// TIA Portal V15.1 export
// export: Created 2024-06-21T08:40:43.8980344Z, ExportSetting WithDefaults, DisplayName Totally Integrated Automation Portal, DisplayVersion V15.1 Update 5, DisplayName TIA Portal Openness, DisplayVersion V15.1 Update 5, DisplayName SINAMICS Startdrive Advanced, DisplayVersion V15.1, DisplayName G130, G150, S120, S150, SINAMICS MV, S210, DisplayVersion V15.1, DisplayName G110M, G120, G120C, G120D, G120P, DisplayVersion V15.1, DisplayName STEP 7 Professional, DisplayVersion V15.1 Update 5, DisplayName STEP 7 Safety, DisplayVersion V15.1, DisplayName WinCC Professional, DisplayVersion V15.1 Update 5, DisplayName SIMATIC Visualization Architect, DisplayVersion V15.1
DATA_BLOCK "_209210ZS01AEAK"   // DB321
{ S7_Optimized_Access := 'FALSE' }
AUTHOR : VCC
VERSION : 0.1
// stored: AutoNumber false, DBAccessibleFromOPCUA true, IsOnlyStoredInLoadMemory false, IsWriteProtectedInAS false
   VAR RETAIN
      AB_AK01E1QM10 { ExternalAccessible := 'False'; ExternalVisible := 'False'; ExternalWritable := 'False'} : Bool;   // 400VAC - Overload protection MoviDrive chain Mode Zone 210
      AB_AK01E1QM11 { ExternalAccessible := 'False'; ExternalVisible := 'False'; ExternalWritable := 'False'} : Bool;   // 400VAC - Overload protection MoviFit chain Mode Zone 210
      AB_AK03E1QM130 { ExternalAccessible := 'False'; ExternalVisible := 'False'; ExternalWritable := 'False'} : Bool;   // 400VAC - Overload protection Brake Resistor 209210CR21
      AB_AK03E1QM133 { ExternalAccessible := 'False'; ExternalVisible := 'False'; ExternalWritable := 'False'} : Bool;   // 400VAC - Overload protection Brake Resistor 209210CR23
      AA_AE01E3FS07_CH1 { ExternalAccessible := 'False'; ExternalVisible := 'False'; ExternalWritable := 'False'} : Bool;   // 24VDC Fuse - ModeZone210 - Switch / Busnode 210AX01 & 210AS10
      AA_AE01E3FS07_CH2 { ExternalAccessible := 'False'; ExternalVisible := 'False'; ExternalWritable := 'False'} : Bool;   // 24VDC Fuse - ModeZone210 - Busnode 210AX02 & 210AS11 & 210AS20
      AC_AE01E3FS08_CH1 { ExternalAccessible := 'False'; ExternalVisible := 'False'; ExternalWritable := 'False'} : Bool;   // 24VDC Fuse - ModeZone210 - RFID Reader
      AA_AE01E3FS08_CH2 { ExternalAccessible := 'False'; ExternalVisible := 'False'; ExternalWritable := 'False'} : Bool;   // 24VDC Fuse - ModeZone210 - Eco Modules
      AD_AE01E3FS07_CH1 { ExternalAccessible := 'False'; ExternalVisible := 'False'; ExternalWritable := 'False'} : Bool;   // 24VDC Fuse - ModeZone210 - Switch / Busnode 210AX01 & 210AS10
      AD_AE01E3FS07_CH2 { ExternalAccessible := 'False'; ExternalVisible := 'False'; ExternalWritable := 'False'} : Bool;   // 24VDC Fuse - ModeZone210 - Busnode 210AX02 & 210AS11 & 210AS20
      AD_AE01E3FS08_CH1 { ExternalAccessible := 'False'; ExternalVisible := 'False'; ExternalWritable := 'False'} : Bool;   // 24VDC Fuse - ModeZone210 - RFID Reader
      AD_AE01E3FS08_CH2 { ExternalAccessible := 'False'; ExternalVisible := 'False'; ExternalWritable := 'False'} : Bool;   // 24VDC Fuse - ModeZone210 - Eco Modules
      AB_AK02E3FS55_CH1 { ExternalAccessible := 'False'; ExternalVisible := 'False'; ExternalWritable := 'False'} : Bool;   // 24VDC Fuse - General - Movidrives AK03 Mode Zone 210
      AA_AK02E3FS100_CH1 { ExternalAccessible := 'False'; ExternalVisible := 'False'; ExternalWritable := 'False'} : Bool;   // 24VDC Fuse - ModeZone 210 - DI/DO 210AX01 & 210AS10
      AA_AK02E3FS100_CH2 { ExternalAccessible := 'False'; ExternalVisible := 'False'; ExternalWritable := 'False'} : Bool;   // 24VDC Fuse - ModeZone 210 - DI/DO 210AX02 & 210AS11 & 210AS20
      AA_AK02E3FS101_CH1 { ExternalAccessible := 'False'; ExternalVisible := 'False'; ExternalWritable := 'False'} : Bool;   // 24VDC Fuse - ModeZone 210 - F-DI/F-DO 210AX01 & 210AS10
      AA_AK02E3FS101_CH2 { ExternalAccessible := 'False'; ExternalVisible := 'False'; ExternalWritable := 'False'} : Bool;   // 24VDC Fuse - ModeZone 210 - F-DI/F-DO 210AX02 & 210AS11 & 210AS20
      AB_AK02E3FS103_CH1 { ExternalAccessible := 'False'; ExternalVisible := 'False'; ExternalWritable := 'False'} : Bool;   // 24VDC Fuse - ModeZone 210 - Movifit Chain 1
      AD_AK02E3FS55_CH1 { ExternalAccessible := 'False'; ExternalVisible := 'False'; ExternalWritable := 'False'} : Bool;   // 24VDC Fuse - General - Movidrives AK03 Mode Zone 210
      AD_AK02E3FS100_CH1 { ExternalAccessible := 'False'; ExternalVisible := 'False'; ExternalWritable := 'False'} : Bool;   // 24VDC Fuse - ModeZone 210 - DI/DO 210AX01 & 210AS10
      AD_AK02E3FS100_CH2 { ExternalAccessible := 'False'; ExternalVisible := 'False'; ExternalWritable := 'False'} : Bool;   // 24VDC Fuse - ModeZone 210 - DI/DO 210AX02 & 210AS11 & 210AS20
      AD_AK02E3FS101_CH1 { ExternalAccessible := 'False'; ExternalVisible := 'False'; ExternalWritable := 'False'} : Bool;   // 24VDC Fuse - ModeZone 210 - F-DI/F-DO 210AX01 & 210AS10
      AD_AK02E3FS101_CH2 { ExternalAccessible := 'False'; ExternalVisible := 'False'; ExternalWritable := 'False'} : Bool;   // 24VDC Fuse - ModeZone 210 - F-DI/F-DO 210AX02 & 210AS11 & 210AS20
      AD_AK02E3FS103_CH1 { ExternalAccessible := 'False'; ExternalVisible := 'False'; ExternalWritable := 'False'} : Bool;   // 24VDC Fuse - ModeZone 210 - Movifit Chain 1
      AK01E1QM10AlarmABCondition { ExternalAccessible := 'False'; ExternalVisible := 'False'; ExternalWritable := 'False'} : Bool;   // Alarm AB condition
      AK01E1QM11AlarmABCondition { ExternalAccessible := 'False'; ExternalVisible := 'False'; ExternalWritable := 'False'} : Bool;   // Alarm AB condition
      AK03E1QM130AlarmABCondition { ExternalAccessible := 'False'; ExternalVisible := 'False'; ExternalWritable := 'False'} : Bool;   // Alarm AB condition
      AK03E1QM133AlarmABCondition { ExternalAccessible := 'False'; ExternalVisible := 'False'; ExternalWritable := 'False'} : Bool;   // Alarm AB condition
      AE01E3FS07_CH1AlarmABCondition { ExternalAccessible := 'False'; ExternalVisible := 'False'; ExternalWritable := 'False'} : Bool;   // Alarm AB condition
      AE01E3FS07_CH2AlarmABCondition { ExternalAccessible := 'False'; ExternalVisible := 'False'; ExternalWritable := 'False'} : Bool;   // Alarm AB condition
      AE01E3FS08_CH2AlarmABCondition { ExternalAccessible := 'False'; ExternalVisible := 'False'; ExternalWritable := 'False'} : Bool;   // Alarm AB condition
      AK02E3FS55_CH1AlarmABCondition { ExternalAccessible := 'False'; ExternalVisible := 'False'; ExternalWritable := 'False'} : Bool;   // Alarm AB condition
      AK02E3FS100_CH1AlarmABCondition { ExternalAccessible := 'False'; ExternalVisible := 'False'; ExternalWritable := 'False'} : Bool;   // Alarm AB condition
      AK02E3FS100_CH2AlarmABCondition { ExternalAccessible := 'False'; ExternalVisible := 'False'; ExternalWritable := 'False'} : Bool;   // Alarm AB condition
      AK02E3FS101_CH1AlarmABCondition { ExternalAccessible := 'False'; ExternalVisible := 'False'; ExternalWritable := 'False'} : Bool;   // Alarm AB condition
      AK02E3FS101_CH2AlarmABCondition { ExternalAccessible := 'False'; ExternalVisible := 'False'; ExternalWritable := 'False'} : Bool;   // Alarm AB condition
      AK02E3FS103_CH1AlarmABCondition { ExternalAccessible := 'False'; ExternalVisible := 'False'; ExternalWritable := 'False'} : Bool;   // Alarm AB condition
      H_209000AK01E1QM10IAnim : Word;   // HMI Animation of the icon
      H_209000AK01E1QM11IAnim : Word;   // HMI Animation of the icon
      H_209000AK03E1QM130IAnim : Word;   // HMI Animation of the icon
      H_209000AK03E1QM133IAnim : Word;   // HMI Animation of the icon
      H_209000AE01E3FS07_CH1IAnim : Word;   // HMI Animation of the icon
      H_209000AE01E3FS07_CH2IAnim : Word;   // HMI Animation of the icon
      H_209000AE01E3FS08_CH1IAnim : Word;   // HMI Animation of the icon
      H_209000AE01E3FS08_CH2IAnim : Word;   // HMI Animation of the icon
      H_209000AK02E3FS55_CH1IAnim : Word;   // HMI Animation of the icon
      H_209000AK02E3FS100_CH1IAnim : Word;   // HMI Animation of the icon
      H_209000AK02E3FS100_CH2IAnim : Word;   // HMI Animation of the icon
      H_209000AK02E3FS101_CH1IAnim : Word;   // HMI Animation of the icon
      H_209000AK02E3FS101_CH2IAnim : Word;   // HMI Animation of the icon
      H_209000AK02E3FS102_CH1IAnim : Word;   // HMI Animation of the icon
      H_209000AK02E3FS102_CH2IAnim : Word;   // HMI Animation of the icon
      H_209000AK02E3FS103_CH1IAnim : Word;   // HMI Animation of the icon
      H_209000AK02E3FS103_CH2IAnim : Word;   // HMI Animation of the icon
      H_DBnr : Int;   // DB number
      H_Anim : Word;   // Animation
      AlarmA { ExternalAccessible := 'False'; ExternalVisible := 'False'; ExternalWritable := 'False'} : Bool;   // Alarm A
      AlarmB { ExternalAccessible := 'False'; ExternalVisible := 'False'; ExternalWritable := 'False'} : Bool;   // Alarm B
      AlarmC { ExternalAccessible := 'False'; ExternalVisible := 'False'; ExternalWritable := 'False'} : Bool;   // Alarm C
      AlarmD { ExternalAccessible := 'False'; ExternalVisible := 'False'; ExternalWritable := 'False'} : Bool;   // Alarm D
      AlarmABCondition { ExternalAccessible := 'False'; ExternalVisible := 'False'; ExternalWritable := 'False'} : Bool;   // Alarm AB condition
   END_VAR
BEGIN
END_DATA_BLOCK
